Omron CX-Programmer project 新工程 (CX-Programmer 9.62)

# PLC 新PLC1: CP1L-E EM

## Global symbols (name address type ; comment)
0.08 BOOL  ; 轴1正转极限
0.09 BOOL  ; 轴1反转极限
0.10 BOOL  ; 轴2正转极限
0.11 BOOL  ; 轴2反转极限
100.04 BOOL  ; 轴1伺服ON
100.05 BOOL  ; 轴2伺服ON
101.00 BOOL  ; 电磁阀1
101.02 BOOL  ; 电磁阀1
101.04 BOOL  ; 蜂鸣器
1.00 BOOL  ; 启动1
1.01 BOOL  ; 启动2
1.02 BOOL  ; 暂停
1.03 BOOL  ; 急停
1.04 BOOL  ; 负压表
1.05 BOOL  ; 光栅
A280.03 BOOL  ; 轴1脉冲输出结束
A280.05 BOOL  ; 轴1无原点标志
A281.03 BOOL  ; 轴3脉冲输出结束
A281.05 BOOL  ; 轴2无原点标志
D0 CHANNEL  ; 轴1定位参数起始
D12 CHANNEL  ; 轴2频率
D14 CHANNEL  ; 轴2脉冲数
D16 CHANNEL  ; 轴2点动频率
D18 CHANNEL  ; 轴2当前值
D2 CHANNEL  ; 轴1频率
D4 CHANNEL  ; 轴1脉冲数
D50 CHANNEL  ; 轴2频率
D6 CHANNEL  ; 轴1点动频率
D8 CHANNEL  ; 轴1当前值
H0 CHANNEL  ; 轴1原点回归速度
H10 CHANNEL  ; 轴1位置1
H12 CHANNEL  ; 轴1位置2
H2 CHANNEL  ; 轴1爬行速度
H4 CHANNEL  ; 轴1运行频率
H50 CHANNEL  ; 轴2原点回归速度
H52 CHANNEL  ; 轴2爬行速度
H54 CHANNEL  ; 轴2运行速度
H56 CHANNEL  ; 轴2调试速度
H58 CHANNEL  ; 轴2原点值
H6 CHANNEL  ; 轴1调试速度
H60 CHANNEL  ; 轴2位置1
H62 CHANNEL  ; 轴2位置2
H64 CHANNEL  ; 轴2位置3
H68 CHANNEL  ; 轴2点胶上抬速度
H8 CHANNEL  ; 轴1原点值
H80 CHANNEL  ; 点胶时间
H82 CHANNEL  ; 产量
W0.00 BOOL  ; 复位步
W0.01 BOOL  ; 等待启动步
W0.02 BOOL  ; 工作步
W0.10 BOOL  ; 调试步
W0.11 BOOL  ; 调试复位步
W103.10 BOOL  ; 点胶动作完成
W10.00 BOOL  ; 轴1正向点动
W10.01 BOOL  ; 轴1反向点动
W10.02 BOOL  ; 轴1停止
W10.03 BOOL  ; 轴1驱动
W10.04 BOOL  ; 轴1定位完成
W10.05 BOOL  ; 轴1原点设置值
W10.06 BOOL  ; 轴1设为原点完成
W11.00 BOOL  ; 轴2正向点动
W11.01 BOOL  ; 轴2反向点动
W11.02 BOOL  ; 轴2停止
W11.03 BOOL  ; 轴2驱动
W11.04 BOOL  ; 轴2定位完成
W11.05 BOOL  ; 轴2设为原点
W11.06 BOOL  ; 轴2设为原点完成
W12.00 BOOL  ; 轴1停止
W12.01 BOOL  ; 轴2停止
W300.00 BOOL  ; 急停
W300.01 BOOL  ; 暂停
W300.02 BOOL  ; 轴1已回原点
W300.03 BOOL  ; 轴2已回原点
W400.00 BOOL  ; 【触摸屏】调试
W400.01 BOOL  ; 轴1+
W400.02 BOOL  ; 轴1-
W400.03 BOOL  ; 轴2+
W400.04 BOOL  ; 轴2-
W5.00 BOOL  ; 急停步

## Program 新程序1 (cyclic task 0)

### Section 段1

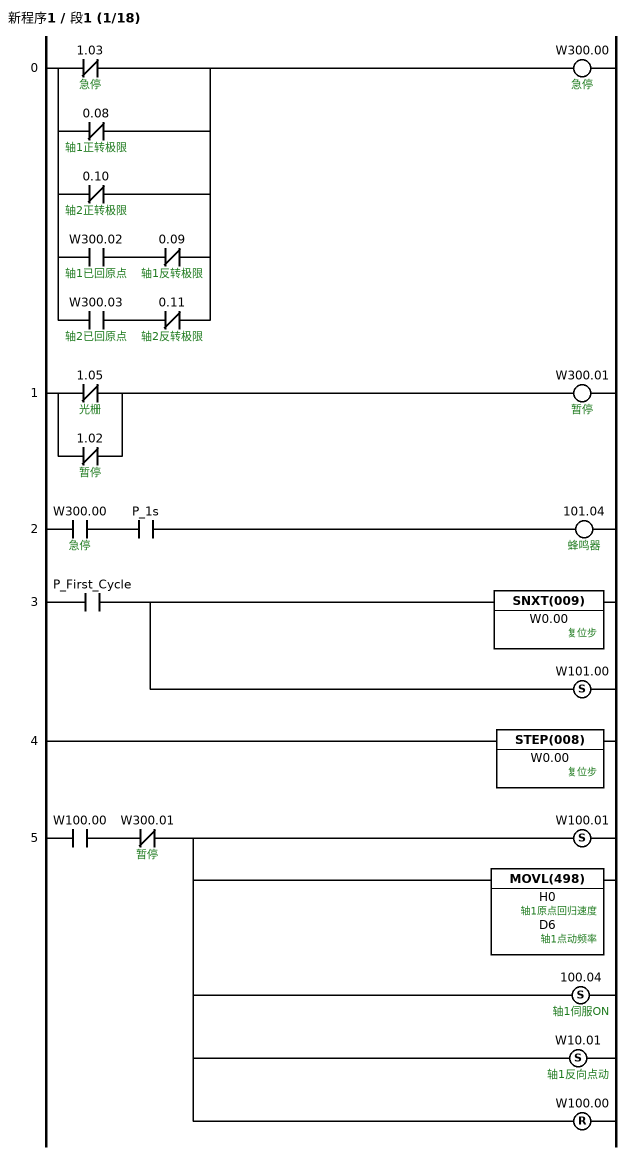
; rung 0
LDNOT 1.03  ; 急停
ORNOT 0.08  ; 轴1正转极限
ORNOT 0.10  ; 轴2正转极限
LD W300.02  ; 轴1已回原点
ANDNOT 0.09  ; 轴1反转极限
ORLD
LD W300.03  ; 轴2已回原点
ANDNOT 0.11  ; 轴2反转极限
ORLD
OUT W300.00  ; 急停
; rung 1
LDNOT 1.05  ; 光栅
ORNOT 1.02  ; 暂停
OUT W300.01  ; 暂停
; rung 2
LD W300.00  ; 急停
AND P_1s
OUT 101.04  ; 蜂鸣器
; rung 3
LD P_First_Cycle
SNXT(009) W0.00  ; 复位步
SET W101.00
; rung 4
STEP(008) W0.00  ; 复位步
; rung 5
LD W100.00
ANDNOT W300.01  ; 暂停
SET W100.01
MOVL(498) H0 D6  ; 轴1原点回归速度, 轴1点动频率
SET 100.04  ; 轴1伺服ON
SET W10.01  ; 轴1反向点动
RSET W100.00

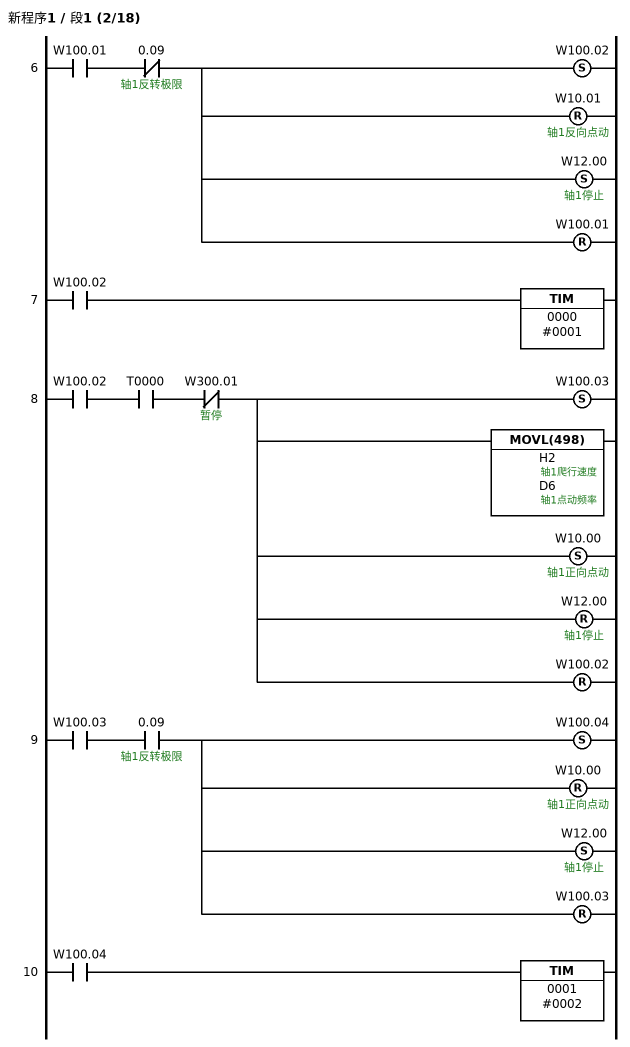
; rung 6
LD W100.01
ANDNOT 0.09  ; 轴1反转极限
SET W100.02
RSET W10.01  ; 轴1反向点动
SET W12.00  ; 轴1停止
RSET W100.01
; rung 7
LD W100.02
TIM 0000 #0001
; rung 8
LD W100.02
AND T0000
ANDNOT W300.01  ; 暂停
SET W100.03
MOVL(498) H2 D6  ; 轴1爬行速度, 轴1点动频率
SET W10.00  ; 轴1正向点动
RSET W12.00  ; 轴1停止
RSET W100.02
; rung 9
LD W100.03
AND 0.09  ; 轴1反转极限
SET W100.04
RSET W10.00  ; 轴1正向点动
SET W12.00  ; 轴1停止
RSET W100.03
; rung 10
LD W100.04
TIM 0001 #0002

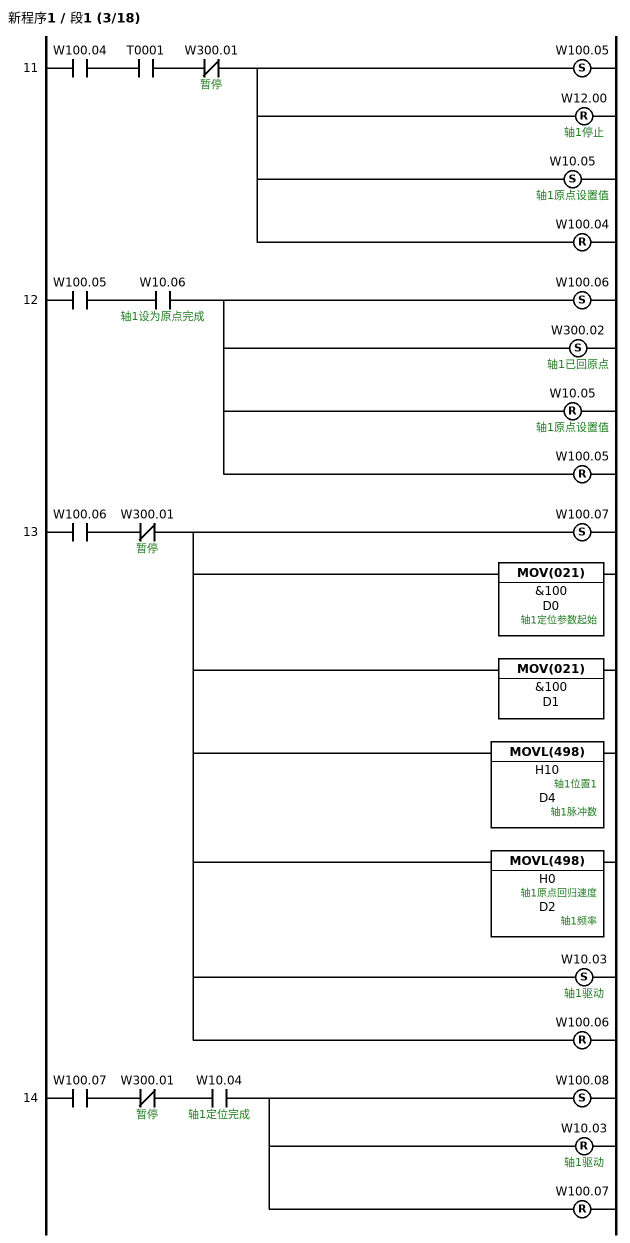
; rung 11
LD W100.04
AND T0001
ANDNOT W300.01  ; 暂停
SET W100.05
RSET W12.00  ; 轴1停止
SET W10.05  ; 轴1原点设置值
RSET W100.04
; rung 12
LD W100.05
AND W10.06  ; 轴1设为原点完成
SET W100.06
SET W300.02  ; 轴1已回原点
RSET W10.05  ; 轴1原点设置值
RSET W100.05
; rung 13
LD W100.06
ANDNOT W300.01  ; 暂停
SET W100.07
MOV(021) &100 D0  ; 轴1定位参数起始
MOV(021) &100 D1
MOVL(498) H10 D4  ; 轴1位置1, 轴1脉冲数
MOVL(498) H0 D2  ; 轴1原点回归速度, 轴1频率
SET W10.03  ; 轴1驱动
RSET W100.06
; rung 14
LD W100.07
ANDNOT W300.01  ; 暂停
AND W10.04  ; 轴1定位完成
SET W100.08
RSET W10.03  ; 轴1驱动
RSET W100.07

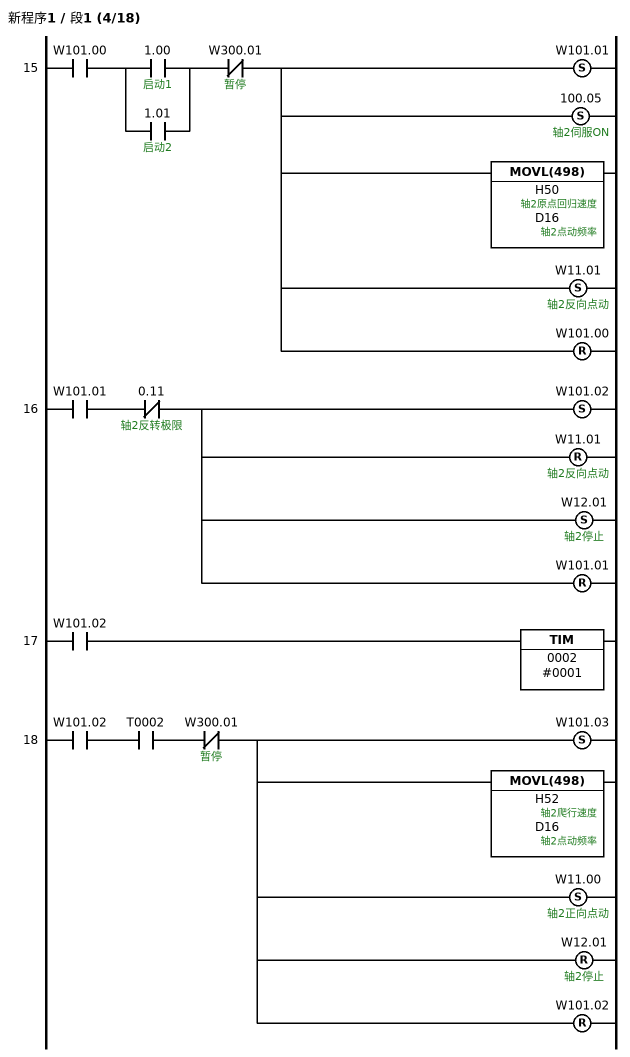
; rung 15
LD W101.00
LD 1.00  ; 启动1
OR 1.01  ; 启动2
ANDLD
ANDNOT W300.01  ; 暂停
SET W101.01
SET 100.05  ; 轴2伺服ON
MOVL(498) H50 D16  ; 轴2原点回归速度, 轴2点动频率
SET W11.01  ; 轴2反向点动
RSET W101.00
; rung 16
LD W101.01
ANDNOT 0.11  ; 轴2反转极限
SET W101.02
RSET W11.01  ; 轴2反向点动
SET W12.01  ; 轴2停止
RSET W101.01
; rung 17
LD W101.02
TIM 0002 #0001
; rung 18
LD W101.02
AND T0002
ANDNOT W300.01  ; 暂停
SET W101.03
MOVL(498) H52 D16  ; 轴2爬行速度, 轴2点动频率
SET W11.00  ; 轴2正向点动
RSET W12.01  ; 轴2停止
RSET W101.02

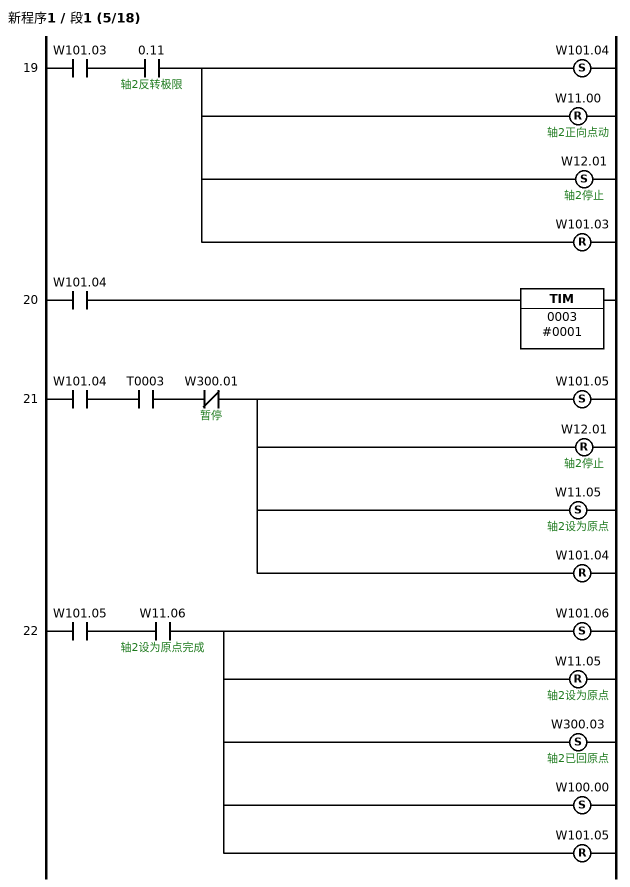
; rung 19
LD W101.03
AND 0.11  ; 轴2反转极限
SET W101.04
RSET W11.00  ; 轴2正向点动
SET W12.01  ; 轴2停止
RSET W101.03
; rung 20
LD W101.04
TIM 0003 #0001
; rung 21
LD W101.04
AND T0003
ANDNOT W300.01  ; 暂停
SET W101.05
RSET W12.01  ; 轴2停止
SET W11.05  ; 轴2设为原点
RSET W101.04
; rung 22
LD W101.05
AND W11.06  ; 轴2设为原点完成
SET W101.06
RSET W11.05  ; 轴2设为原点
SET W300.03  ; 轴2已回原点
SET W100.00
RSET W101.05

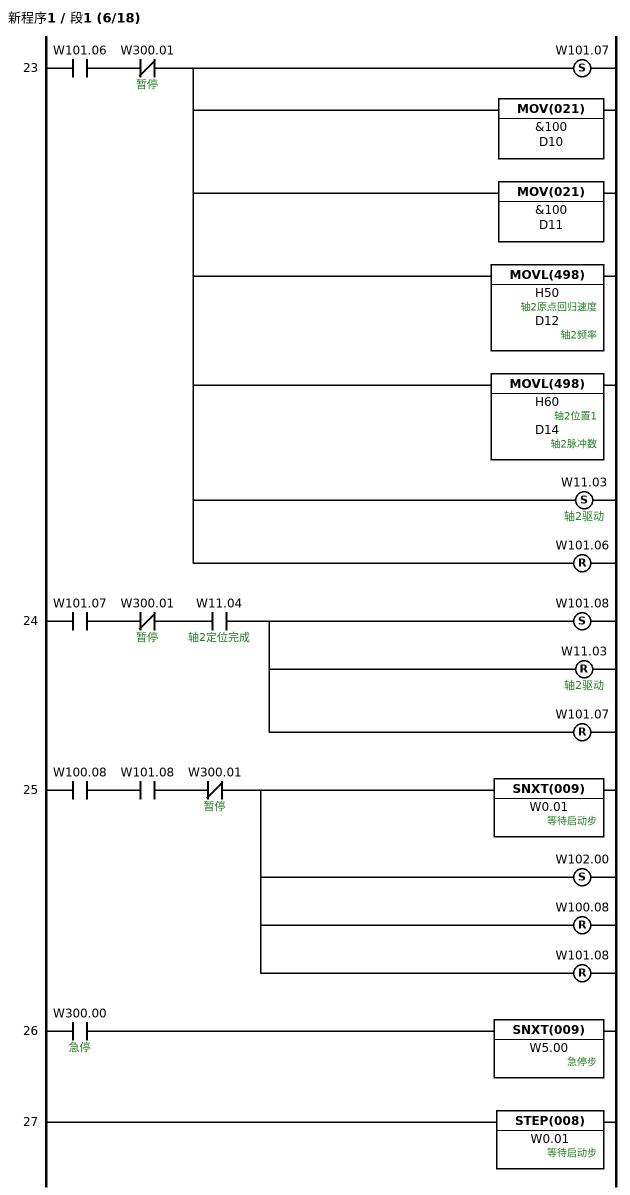
; rung 23
LD W101.06
ANDNOT W300.01  ; 暂停
SET W101.07
MOV(021) &100 D10
MOV(021) &100 D11
MOVL(498) H50 D12  ; 轴2原点回归速度, 轴2频率
MOVL(498) H60 D14  ; 轴2位置1, 轴2脉冲数
SET W11.03  ; 轴2驱动
RSET W101.06
; rung 24
LD W101.07
ANDNOT W300.01  ; 暂停
AND W11.04  ; 轴2定位完成
SET W101.08
RSET W11.03  ; 轴2驱动
RSET W101.07
; rung 25
LD W100.08
AND W101.08
ANDNOT W300.01  ; 暂停
SNXT(009) W0.01  ; 等待启动步
SET W102.00
RSET W100.08
RSET W101.08
; rung 26
LD W300.00  ; 急停
SNXT(009) W5.00  ; 急停步
; rung 27
STEP(008) W0.01  ; 等待启动步

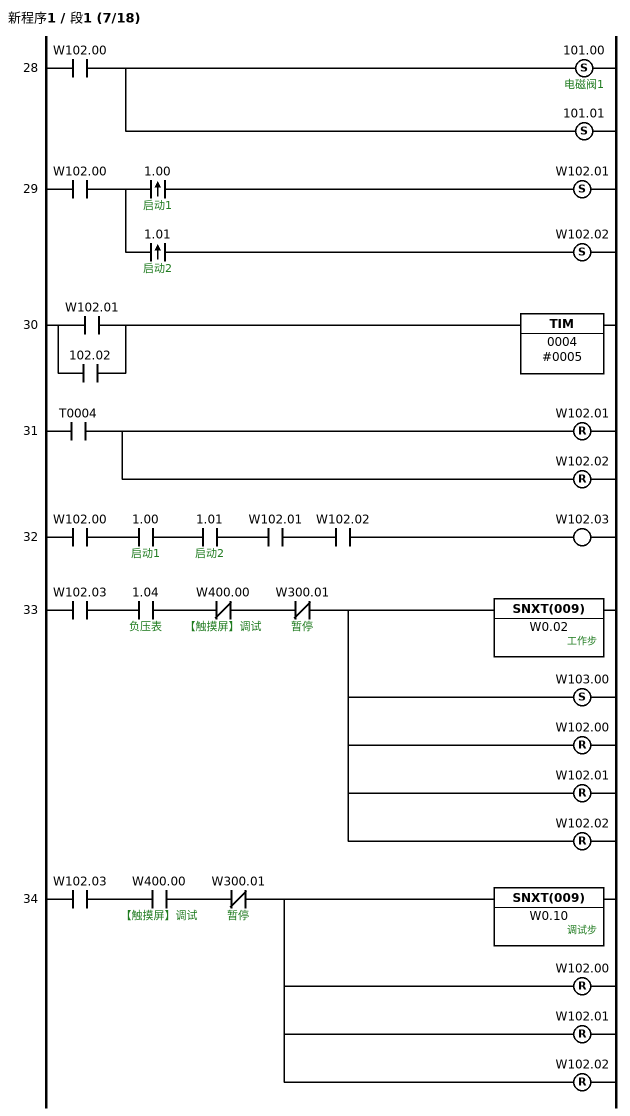
; rung 28
LD W102.00
SET 101.00  ; 电磁阀1
SET 101.01
; rung 29
LD W102.00
OUT TR0
@AND 1.00  ; 启动1
SET W102.01
LD TR0
@AND 1.01  ; 启动2
SET W102.02
; rung 30
LD W102.01
OR 102.02
TIM 0004 #0005
; rung 31
LD T0004
RSET W102.01
RSET W102.02
; rung 32
LD W102.00
AND 1.00  ; 启动1
AND 1.01  ; 启动2
AND W102.01
AND W102.02
OUT W102.03
; rung 33
LD W102.03
AND 1.04  ; 负压表
ANDNOT W400.00  ; 【触摸屏】调试
ANDNOT W300.01  ; 暂停
SNXT(009) W0.02  ; 工作步
SET W103.00
RSET W102.00
RSET W102.01
RSET W102.02
; rung 34
LD W102.03
AND W400.00  ; 【触摸屏】调试
ANDNOT W300.01  ; 暂停
SNXT(009) W0.10  ; 调试步
RSET W102.00
RSET W102.01
RSET W102.02

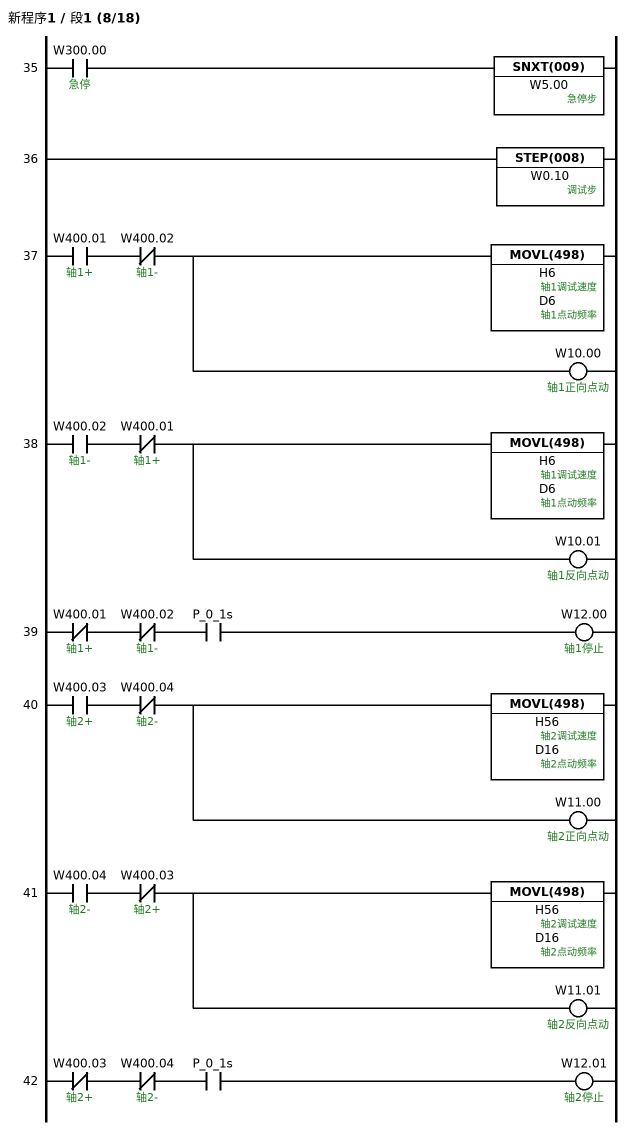
; rung 35
LD W300.00  ; 急停
SNXT(009) W5.00  ; 急停步
; rung 36
STEP(008) W0.10  ; 调试步
; rung 37
LD W400.01  ; 轴1+
ANDNOT W400.02  ; 轴1-
MOVL(498) H6 D6  ; 轴1调试速度, 轴1点动频率
OUT W10.00  ; 轴1正向点动
; rung 38
LD W400.02  ; 轴1-
ANDNOT W400.01  ; 轴1+
MOVL(498) H6 D6  ; 轴1调试速度, 轴1点动频率
OUT W10.01  ; 轴1反向点动
; rung 39
LDNOT W400.01  ; 轴1+
ANDNOT W400.02  ; 轴1-
AND P_0_1s
OUT W12.00  ; 轴1停止
; rung 40
LD W400.03  ; 轴2+
ANDNOT W400.04  ; 轴2-
MOVL(498) H56 D16  ; 轴2调试速度, 轴2点动频率
OUT W11.00  ; 轴2正向点动
; rung 41
LD W400.04  ; 轴2-
ANDNOT W400.03  ; 轴2+
MOVL(498) H56 D16  ; 轴2调试速度, 轴2点动频率
OUT W11.01  ; 轴2反向点动
; rung 42
LDNOT W400.03  ; 轴2+
ANDNOT W400.04  ; 轴2-
AND P_0_1s
OUT W12.01  ; 轴2停止

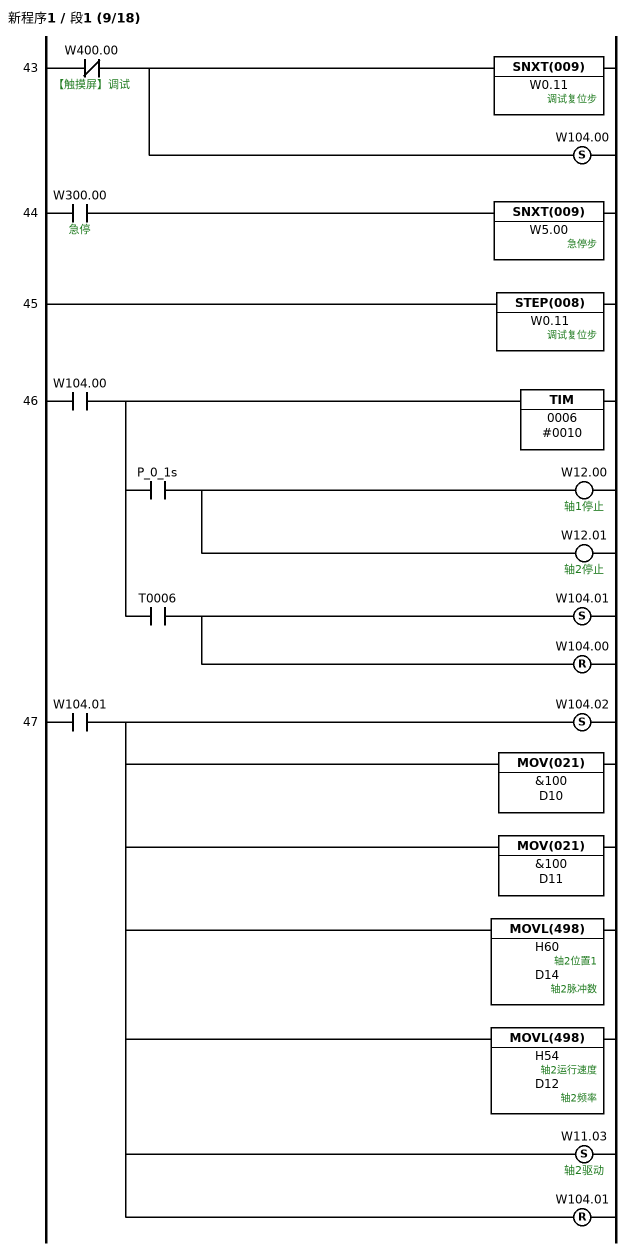
; rung 43
LDNOT W400.00  ; 【触摸屏】调试
SNXT(009) W0.11  ; 调试复位步
SET W104.00
; rung 44
LD W300.00  ; 急停
SNXT(009) W5.00  ; 急停步
; rung 45
STEP(008) W0.11  ; 调试复位步
; rung 46
LD W104.00
OUT TR0
TIM 0006 #0010
AND P_0_1s
OUT W12.00  ; 轴1停止
OUT W12.01  ; 轴2停止
LD TR0
AND T0006
SET W104.01
RSET W104.00
; rung 47
LD W104.01
SET W104.02
MOV(021) &100 D10
MOV(021) &100 D11
MOVL(498) H60 D14  ; 轴2位置1, 轴2脉冲数
MOVL(498) H54 D12  ; 轴2运行速度, 轴2频率
SET W11.03  ; 轴2驱动
RSET W104.01

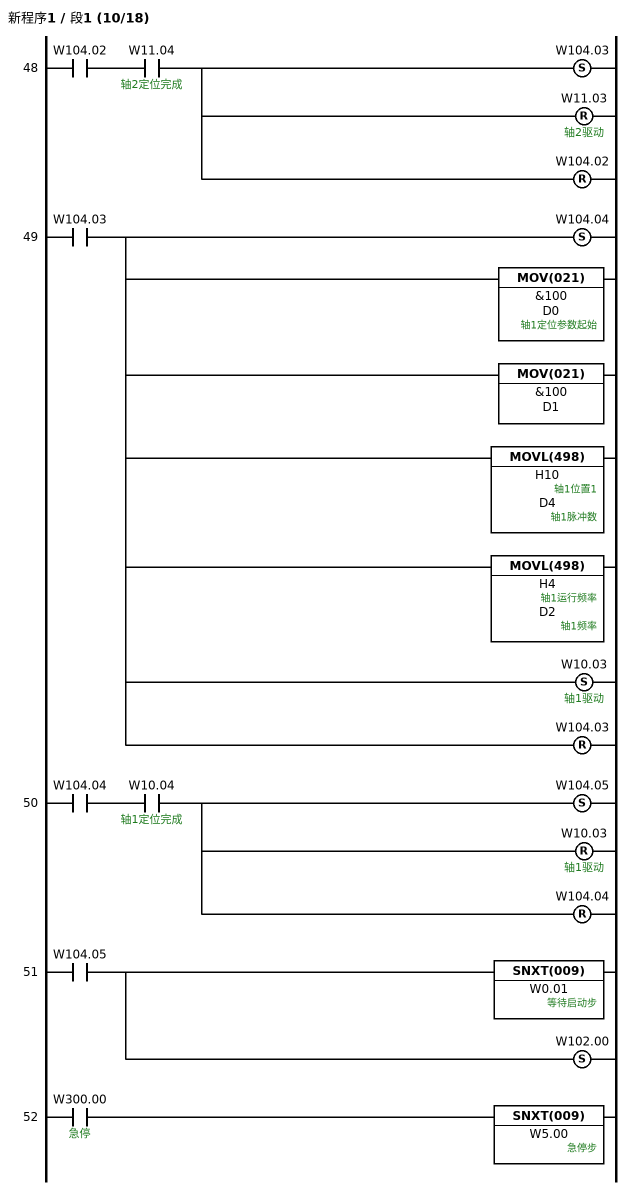
; rung 48
LD W104.02
AND W11.04  ; 轴2定位完成
SET W104.03
RSET W11.03  ; 轴2驱动
RSET W104.02
; rung 49
LD W104.03
SET W104.04
MOV(021) &100 D0  ; 轴1定位参数起始
MOV(021) &100 D1
MOVL(498) H10 D4  ; 轴1位置1, 轴1脉冲数
MOVL(498) H4 D2  ; 轴1运行频率, 轴1频率
SET W10.03  ; 轴1驱动
RSET W104.03
; rung 50
LD W104.04
AND W10.04  ; 轴1定位完成
SET W104.05
RSET W10.03  ; 轴1驱动
RSET W104.04
; rung 51
LD W104.05
SNXT(009) W0.01  ; 等待启动步
SET W102.00
; rung 52
LD W300.00  ; 急停
SNXT(009) W5.00  ; 急停步

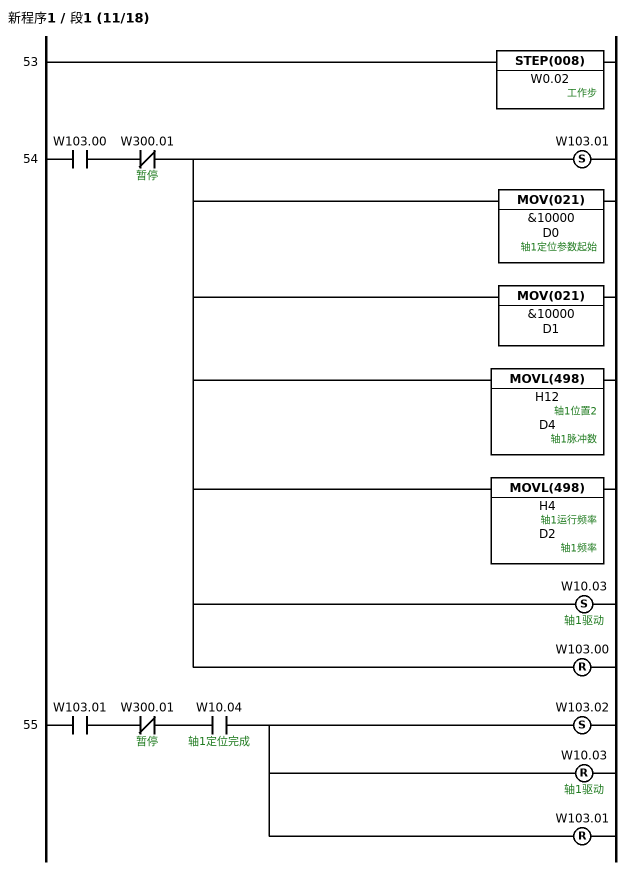
; rung 53
STEP(008) W0.02  ; 工作步
; rung 54
LD W103.00
ANDNOT W300.01  ; 暂停
SET W103.01
MOV(021) &10000 D0  ; 轴1定位参数起始
MOV(021) &10000 D1
MOVL(498) H12 D4  ; 轴1位置2, 轴1脉冲数
MOVL(498) H4 D2  ; 轴1运行频率, 轴1频率
SET W10.03  ; 轴1驱动
RSET W103.00
; rung 55
LD W103.01
ANDNOT W300.01  ; 暂停
AND W10.04  ; 轴1定位完成
SET W103.02
RSET W10.03  ; 轴1驱动
RSET W103.01

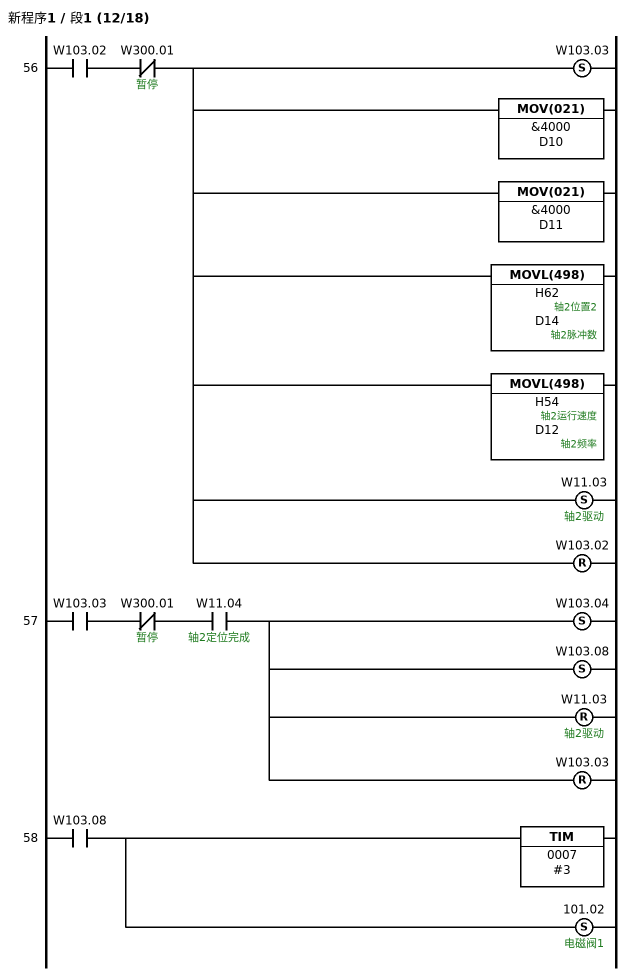
; rung 56
LD W103.02
ANDNOT W300.01  ; 暂停
SET W103.03
MOV(021) &4000 D10
MOV(021) &4000 D11
MOVL(498) H62 D14  ; 轴2位置2, 轴2脉冲数
MOVL(498) H54 D12  ; 轴2运行速度, 轴2频率
SET W11.03  ; 轴2驱动
RSET W103.02
; rung 57
LD W103.03
ANDNOT W300.01  ; 暂停
AND W11.04  ; 轴2定位完成
SET W103.04
SET W103.08
RSET W11.03  ; 轴2驱动
RSET W103.03
; rung 58
LD W103.08
TIM 0007 #3
SET 101.02  ; 电磁阀1

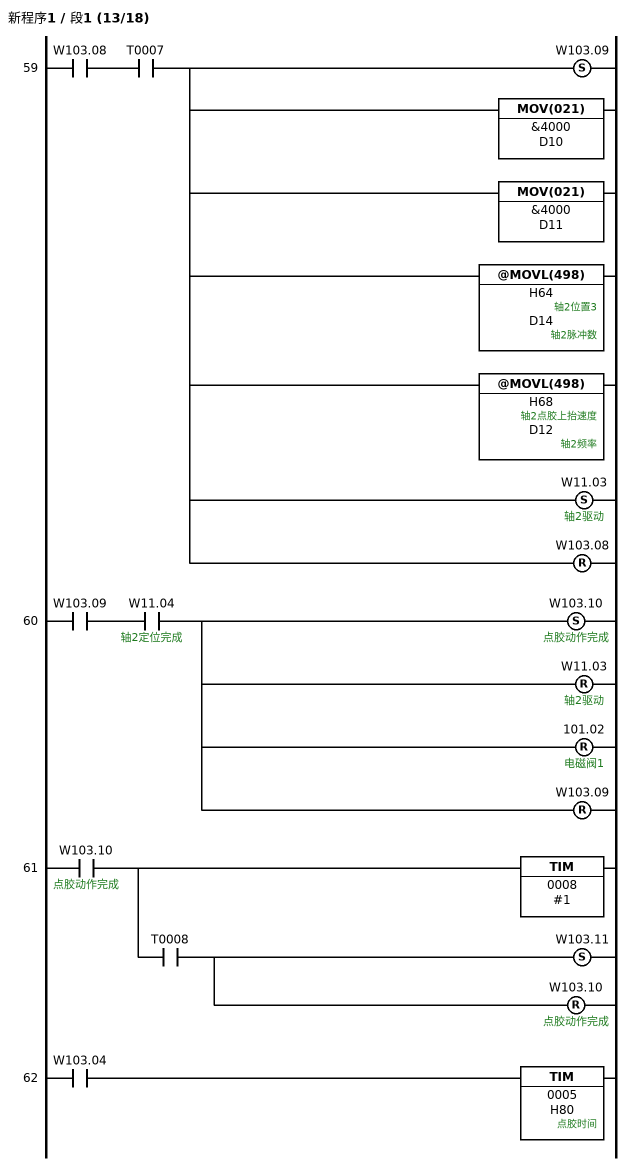
; rung 59
LD W103.08
AND T0007
SET W103.09
MOV(021) &4000 D10
MOV(021) &4000 D11
@MOVL(498) H64 D14  ; 轴2位置3, 轴2脉冲数
@MOVL(498) H68 D12  ; 轴2点胶上抬速度, 轴2频率
SET W11.03  ; 轴2驱动
RSET W103.08
; rung 60
LD W103.09
AND W11.04  ; 轴2定位完成
SET W103.10  ; 点胶动作完成
RSET W11.03  ; 轴2驱动
RSET 101.02  ; 电磁阀1
RSET W103.09
; rung 61
LD W103.10  ; 点胶动作完成
TIM 0008 #1
AND T0008
SET W103.11
RSET W103.10  ; 点胶动作完成
; rung 62
LD W103.04
TIM 0005 H80  ; 点胶时间

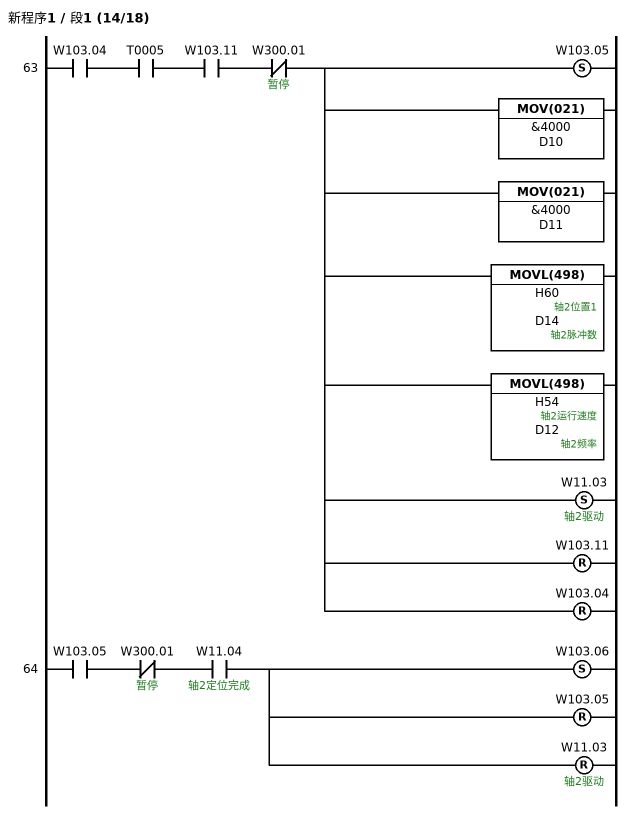
; rung 63
LD W103.04
AND T0005
AND W103.11
ANDNOT W300.01  ; 暂停
SET W103.05
MOV(021) &4000 D10
MOV(021) &4000 D11
MOVL(498) H60 D14  ; 轴2位置1, 轴2脉冲数
MOVL(498) H54 D12  ; 轴2运行速度, 轴2频率
SET W11.03  ; 轴2驱动
RSET W103.11
RSET W103.04
; rung 64
LD W103.05
ANDNOT W300.01  ; 暂停
AND W11.04  ; 轴2定位完成
SET W103.06
RSET W103.05
RSET W11.03  ; 轴2驱动

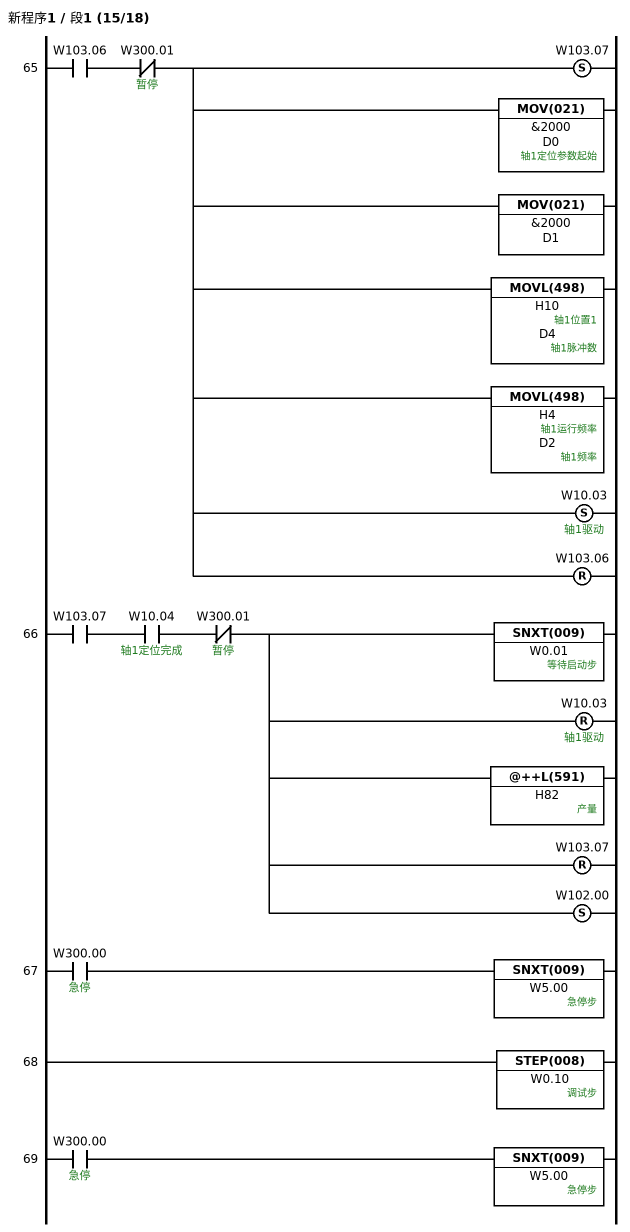
; rung 65
LD W103.06
ANDNOT W300.01  ; 暂停
SET W103.07
MOV(021) &2000 D0  ; 轴1定位参数起始
MOV(021) &2000 D1
MOVL(498) H10 D4  ; 轴1位置1, 轴1脉冲数
MOVL(498) H4 D2  ; 轴1运行频率, 轴1频率
SET W10.03  ; 轴1驱动
RSET W103.06
; rung 66
LD W103.07
AND W10.04  ; 轴1定位完成
ANDNOT W300.01  ; 暂停
SNXT(009) W0.01  ; 等待启动步
RSET W10.03  ; 轴1驱动
@++L(591) H82  ; 产量
RSET W103.07
SET W102.00
; rung 67
LD W300.00  ; 急停
SNXT(009) W5.00  ; 急停步
; rung 68
STEP(008) W0.10  ; 调试步
; rung 69
LD W300.00  ; 急停
SNXT(009) W5.00  ; 急停步

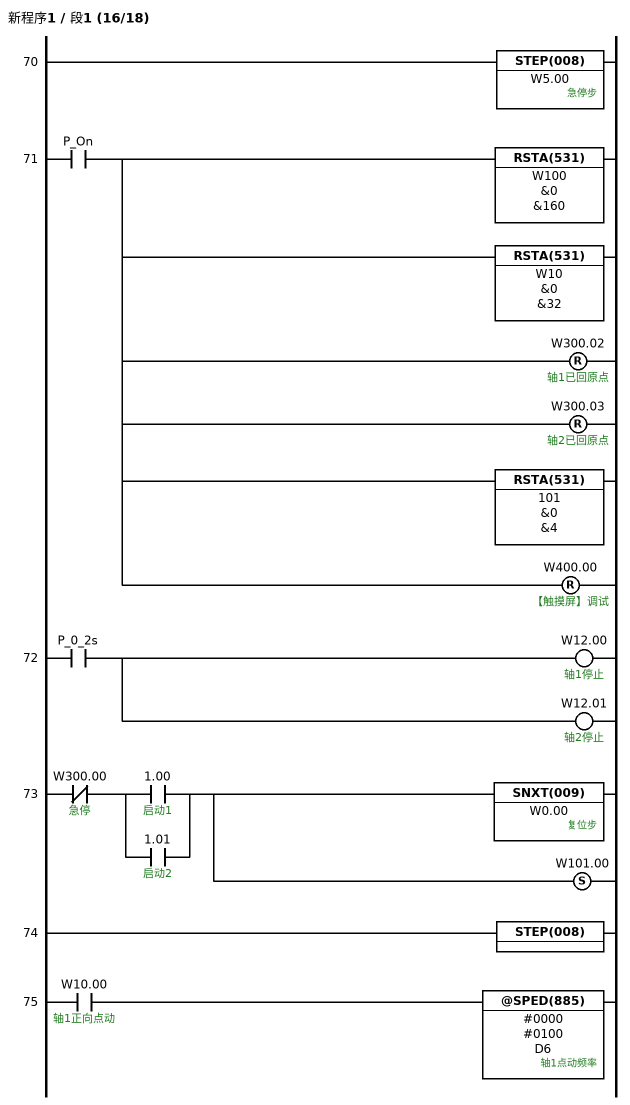
; rung 70
STEP(008) W5.00  ; 急停步
; rung 71
LD P_On
RSTA(531) W100 &0 &160
RSTA(531) W10 &0 &32
RSET W300.02  ; 轴1已回原点
RSET W300.03  ; 轴2已回原点
RSTA(531) 101 &0 &4
RSET W400.00  ; 【触摸屏】调试
; rung 72
LD P_0_2s
OUT W12.00  ; 轴1停止
OUT W12.01  ; 轴2停止
; rung 73
LDNOT W300.00  ; 急停
LD 1.00  ; 启动1
OR 1.01  ; 启动2
ANDLD
SNXT(009) W0.00  ; 复位步
SET W101.00
; rung 74
STEP(008)
; rung 75
LD W10.00  ; 轴1正向点动
@SPED(885) #0000 #0100 D6  ; 轴1点动频率

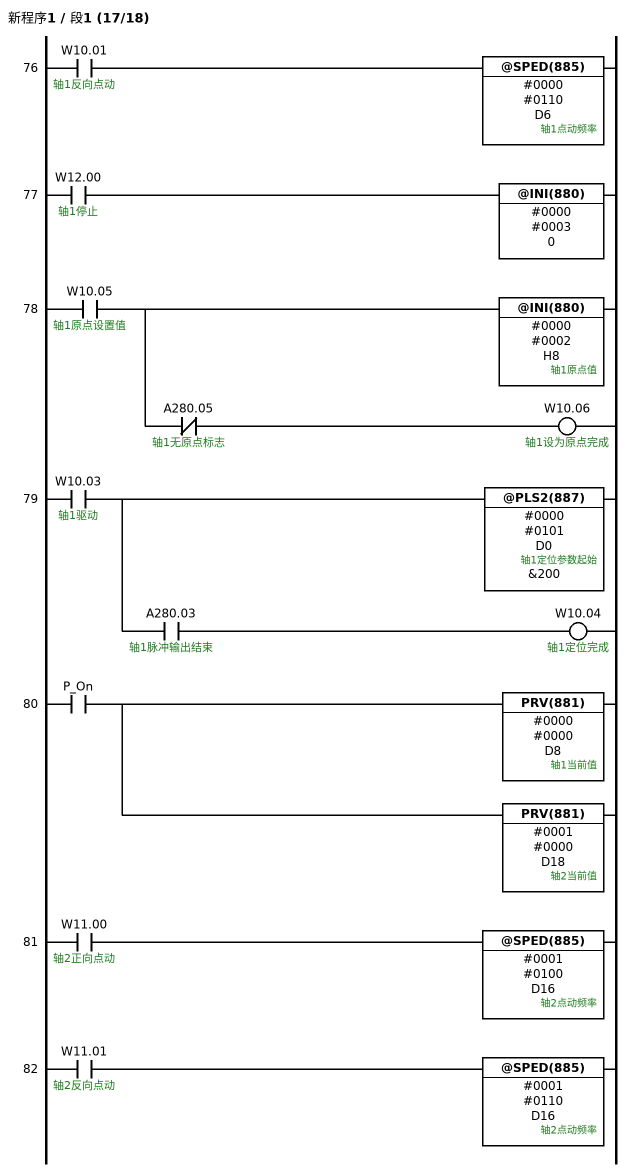
; rung 76
LD W10.01  ; 轴1反向点动
@SPED(885) #0000 #0110 D6  ; 轴1点动频率
; rung 77
LD W12.00  ; 轴1停止
@INI(880) #0000 #0003 0
; rung 78
LD W10.05  ; 轴1原点设置值
@INI(880) #0000 #0002 H8  ; 轴1原点值
ANDNOT A280.05  ; 轴1无原点标志
OUT W10.06  ; 轴1设为原点完成
; rung 79
LD W10.03  ; 轴1驱动
@PLS2(887) #0000 #0101 D0 &200  ; 轴1定位参数起始
AND A280.03  ; 轴1脉冲输出结束
OUT W10.04  ; 轴1定位完成
; rung 80
LD P_On
PRV(881) #0000 #0000 D8  ; 轴1当前值
PRV(881) #0001 #0000 D18  ; 轴2当前值
; rung 81
LD W11.00  ; 轴2正向点动
@SPED(885) #0001 #0100 D16  ; 轴2点动频率
; rung 82
LD W11.01  ; 轴2反向点动
@SPED(885) #0001 #0110 D16  ; 轴2点动频率

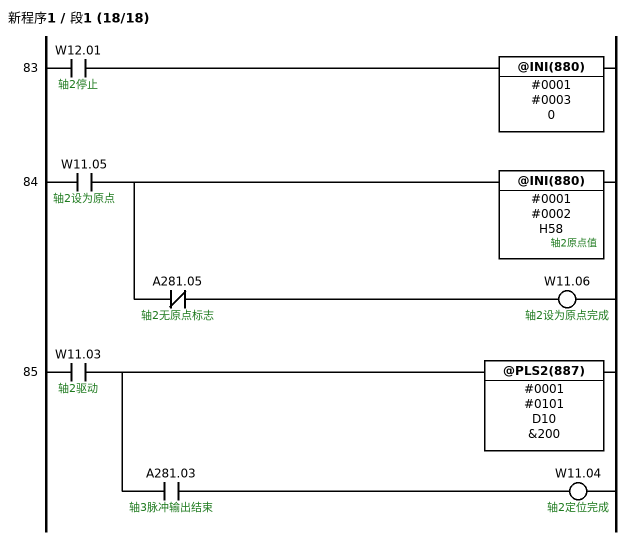
; rung 83
LD W12.01  ; 轴2停止
@INI(880) #0001 #0003 0
; rung 84
LD W11.05  ; 轴2设为原点
@INI(880) #0001 #0002 H58  ; 轴2原点值
ANDNOT A281.05  ; 轴2无原点标志
OUT W11.06  ; 轴2设为原点完成
; rung 85
LD W11.03  ; 轴2驱动
@PLS2(887) #0001 #0101 D10 &200
AND A281.03  ; 轴3脉冲输出结束
OUT W11.04  ; 轴2定位完成

### Section END
; rung 0
END(001)